// TIA Portal V19 export
DATA_BLOCK "DTrk"   // DB134
{ DB_Accessible_From_OPC_UA := 'FALSE' }
// stored: DBAccessibleFromOPCUA false, MemoryReserve 100
   VAR
      Empty : "udt_DTrk";
   END_VAR
   VAR RETAIN
      UNCUT : "udt_DTrk";
      CUTTED : "udt_DTrk";
      LAST_CUTTED : "udt_DTrk";
   END_VAR
BEGIN
END_DATA_BLOCK
